// TIA Portal V21 export
TYPE "LBC_typeMotorStarterConfiguration"
TITLE = LBC_typeMotorStarterConfiguration
// Module related configuration parameters
   STRUCT
      referenceDesignator { S7_SetPoint := 'True'} : WString[25] := WSTRING#'MotorStarter';   // Device name or device ID
      startingControlTime { S7_SetPoint := 'True'} : Time := T#5s;   // Control time for receiving feedback motor is running or time to ramp up motor if feedback is disabled
      stoppingControlTime { S7_SetPoint := 'True'} : Time := T#5s;   // Control time for feedback motor is stopped (fb running has disappeared) or time to ramp down motor if feedback is disabled
      resetTime { S7_SetPoint := 'True'} : Time := T#5s;   // Control time for reset - time to set reset output / the reset signal is present at the reset output (advanced motor starter)
      disableFeedbackRunning { S7_SetPoint := 'True'} : Bool := TRUE;   // Disable feedback for started / running motor
      disableFeedbackError { S7_SetPoint := 'True'} : Bool := TRUE;   // Disable feedback for error monitoring (e.g. over temperature)
      disableAlarms { S7_SetPoint := 'True'} : Bool;   // Disable the alarms of the block
   END_STRUCT;
END_TYPE
